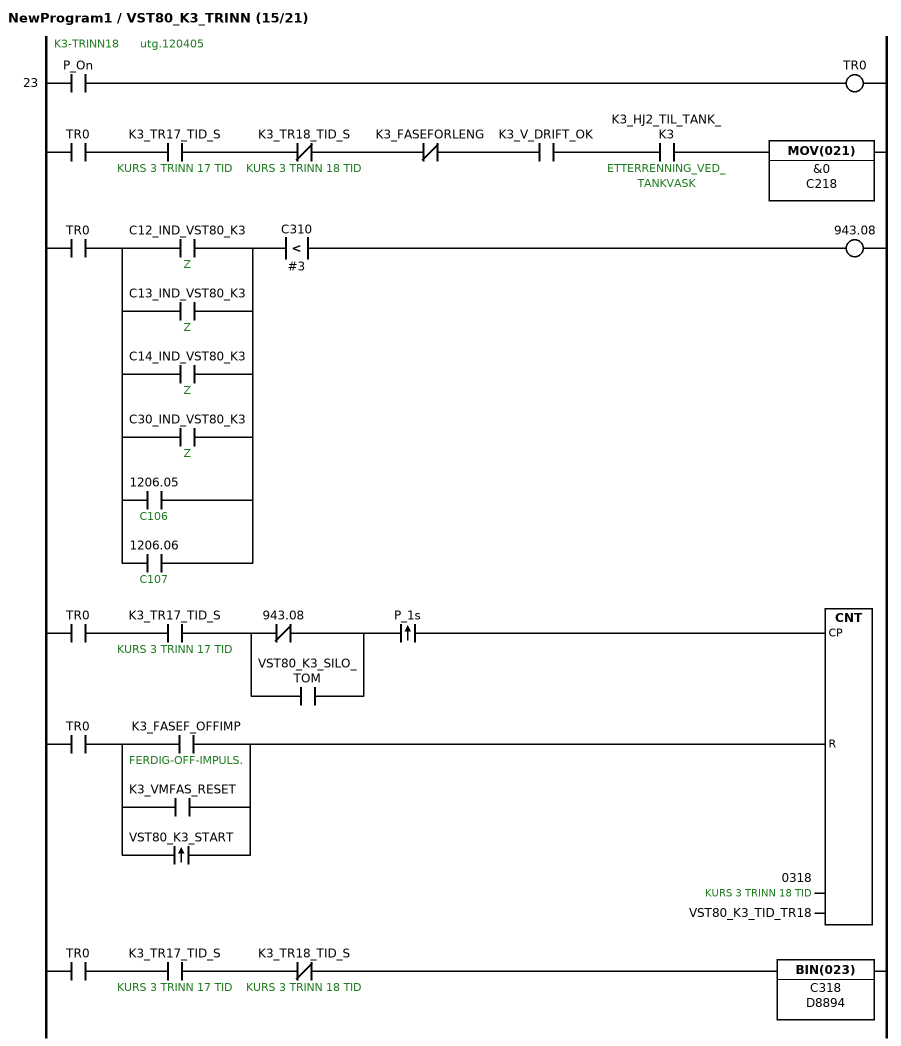
; [picture p336: NewProgram1 / VST80_K3_TRINN, rungs 23-23]
; rung 23: K3-TRINN18      utg.120405
LD P_On
OUT TR0
AND K3_TR17_TID_S  ; KURS 3 TRINN 17 TID
ANDNOT K3_TR18_TID_S  ; KURS 3 TRINN 18 TID
ANDNOT K3_FASEFORLENG
AND K3_V_DRIFT_OK
AND K3_HJ2_TIL_TANK_K3  ; ETTERRENNING_VED_TANKVASK
MOV(021) &0 C218
LD TR0
LD C12_IND_VST80_K3  ; Z
OR C13_IND_VST80_K3  ; Z
OR C14_IND_VST80_K3  ; Z
OR C30_IND_VST80_K3  ; Z
OR 1206.05  ; C106
OR 1206.06  ; C107
ANDLD
AND<(310) C310 #3
OUT 943.08
LD TR0
AND K3_TR17_TID_S  ; KURS 3 TRINN 17 TID
LDNOT 943.08
OR VST80_K3_SILO_TOM
ANDLD
@AND P_1s
LD TR0
LD K3_FASEF_OFFIMP  ; FERDIG-OFF-IMPULS.
OR K3_VMFAS_RESET
@OR VST80_K3_START
ANDLD
CNT 0318 VST80_K3_TID_TR18  ; KURS 3 TRINN 18 TID
LD TR0
AND K3_TR17_TID_S  ; KURS 3 TRINN 17 TID
ANDNOT K3_TR18_TID_S  ; KURS 3 TRINN 18 TID
BIN(023) C318 D8894

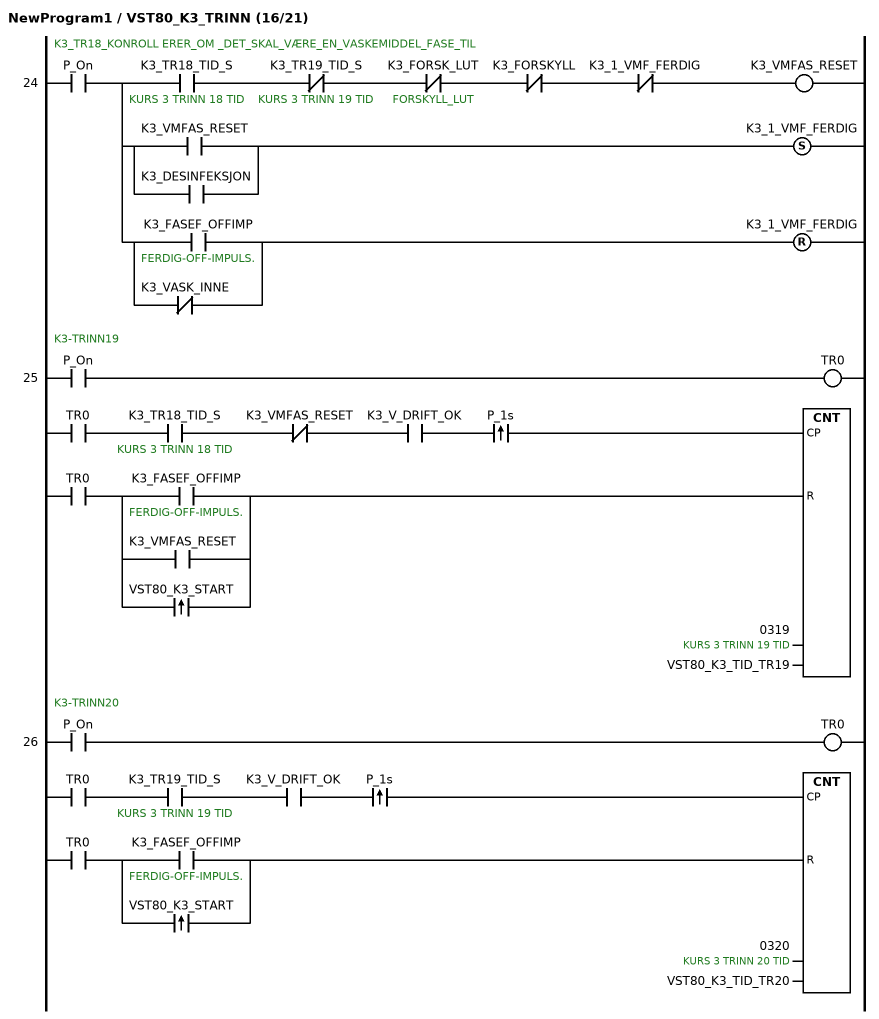
; rung 24: K3_TR18_KONROLL ERER_OM_DET_SKAL_VÆRE_EN_VASKEMIDDEL_FASE_TIL
LD P_On
OUT TR0
AND K3_TR18_TID_S  ; KURS 3 TRINN 18 TID
ANDNOT K3_TR19_TID_S  ; KURS 3 TRINN 19 TID
ANDNOT K3_FORSK_LUT  ; FORSKYLL_LUT
ANDNOT K3_FORSKYLL
ANDNOT K3_1_VMF_FERDIG
OUT K3_VMFAS_RESET
LD TR0
LD K3_VMFAS_RESET
OR K3_DESINFEKSJON
ANDLD
SET K3_1_VMF_FERDIG
LD TR0
LD K3_FASEF_OFFIMP  ; FERDIG-OFF-IMPULS.
ORNOT K3_VASK_INNE
ANDLD
RSET K3_1_VMF_FERDIG
; rung 25: K3-TRINN19
LD P_On
OUT TR0
AND K3_TR18_TID_S  ; KURS 3 TRINN 18 TID
ANDNOT K3_VMFAS_RESET
AND K3_V_DRIFT_OK
@AND P_1s
LD TR0
LD K3_FASEF_OFFIMP  ; FERDIG-OFF-IMPULS.
OR K3_VMFAS_RESET
@OR VST80_K3_START
ANDLD
CNT 0319 VST80_K3_TID_TR19  ; KURS 3 TRINN 19 TID
; rung 26: K3-TRINN20
LD P_On
OUT TR0
AND K3_TR19_TID_S  ; KURS 3 TRINN 19 TID
AND K3_V_DRIFT_OK
@AND P_1s
LD TR0
LD K3_FASEF_OFFIMP  ; FERDIG-OFF-IMPULS.
@OR VST80_K3_START
ANDLD
CNT 0320 VST80_K3_TID_TR20  ; KURS 3 TRINN 20 TID

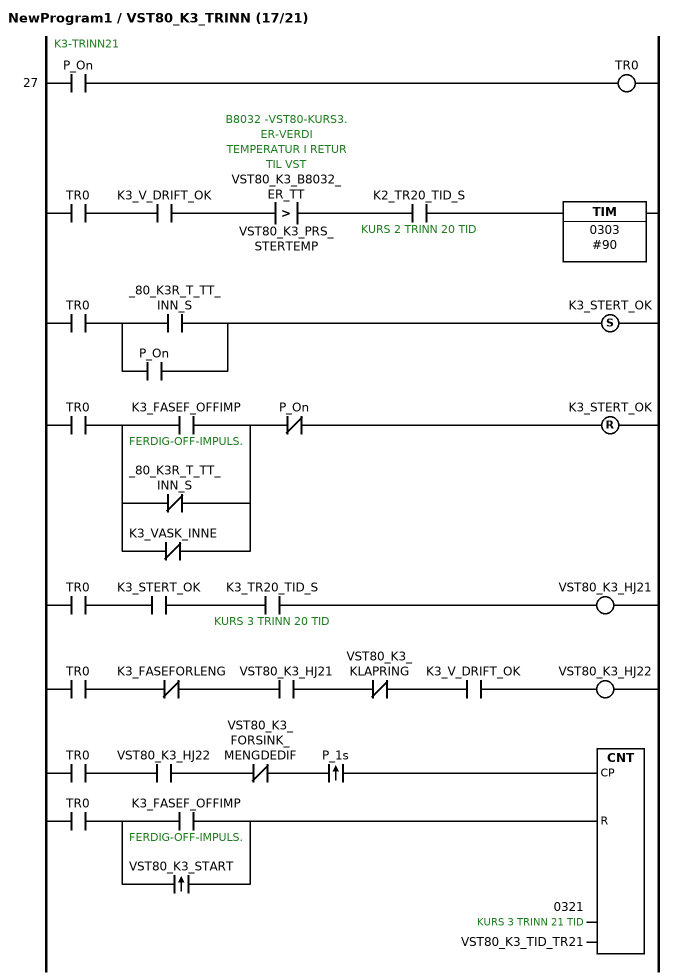
; rung 27: K3-TRINN21
LD P_On
OUT TR0
AND K3_V_DRIFT_OK
AND>(320) VST80_K3_B8032_ER_TT VST80_K3_PRS_STERTEMP  ; B8032 -VST80-KURS3. ER-VERDI TEMPERATUR I RETUR TIL VST
AND K2_TR20_TID_S  ; KURS 2 TRINN 20 TID
TIM 0303 #90
LD TR0
LD _80_K3R_T_TT_INN_S
OR P_On
ANDLD
SET K3_STERT_OK
LD TR0
LD K3_FASEF_OFFIMP  ; FERDIG-OFF-IMPULS.
ORNOT _80_K3R_T_TT_INN_S
ORNOT K3_VASK_INNE
ANDLD
ANDNOT P_On
RSET K3_STERT_OK
LD TR0
AND K3_STERT_OK
AND K3_TR20_TID_S  ; KURS 3 TRINN 20 TID
OUT VST80_K3_HJ21
LD TR0
ANDNOT K3_FASEFORLENG
AND VST80_K3_HJ21
ANDNOT VST80_K3_KLAPRING
AND K3_V_DRIFT_OK
OUT VST80_K3_HJ22
LD TR0
AND VST80_K3_HJ22
ANDNOT VST80_K3_FORSINK_MENGDEDIF
@AND P_1s
LD TR0
LD K3_FASEF_OFFIMP  ; FERDIG-OFF-IMPULS.
@OR VST80_K3_START
ANDLD
CNT 0321 VST80_K3_TID_TR21  ; KURS 3 TRINN 21 TID

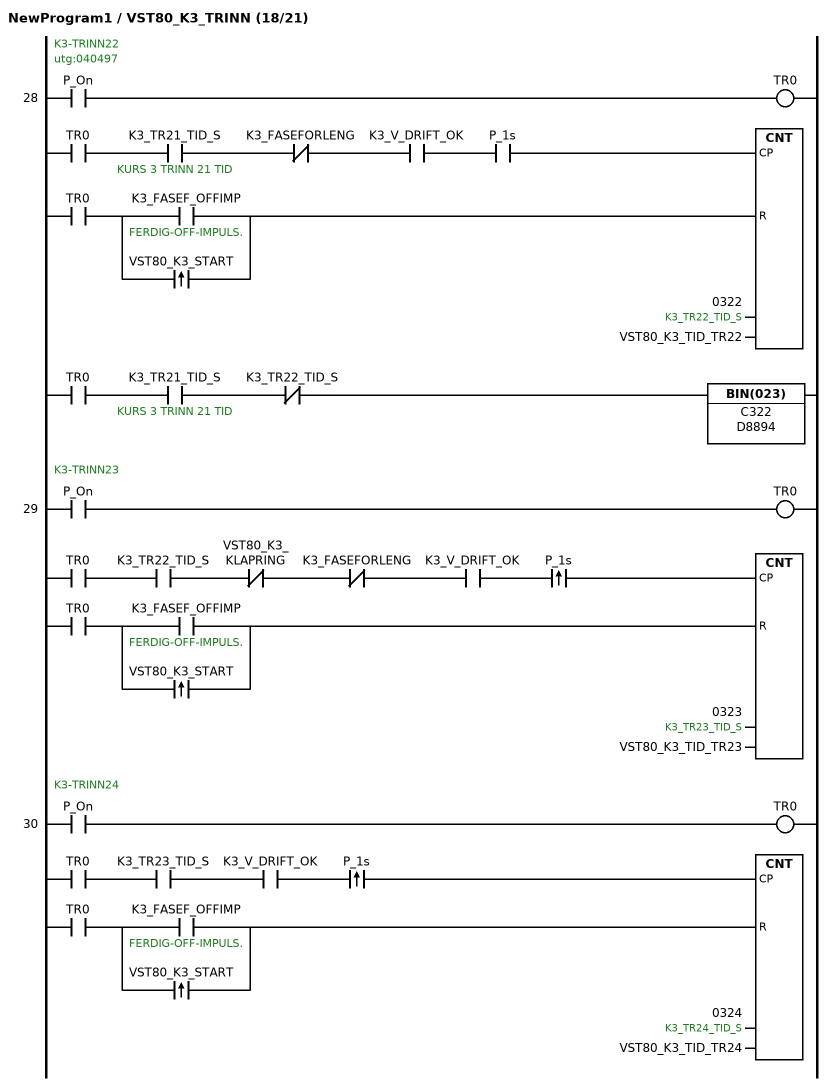
; rung 28: K3-TRINN22 / utg:040497
LD P_On
OUT TR0
AND K3_TR21_TID_S  ; KURS 3 TRINN 21 TID
ANDNOT K3_FASEFORLENG
AND K3_V_DRIFT_OK
AND P_1s
LD TR0
LD K3_FASEF_OFFIMP  ; FERDIG-OFF-IMPULS.
@OR VST80_K3_START
ANDLD
CNT 0322 VST80_K3_TID_TR22  ; K3_TR22_TID_S
LD TR0
AND K3_TR21_TID_S  ; KURS 3 TRINN 21 TID
ANDNOT K3_TR22_TID_S
BIN(023) C322 D8894
; rung 29: K3-TRINN23
LD P_On
OUT TR0
AND K3_TR22_TID_S
ANDNOT VST80_K3_KLAPRING
ANDNOT K3_FASEFORLENG
AND K3_V_DRIFT_OK
@AND P_1s
LD TR0
LD K3_FASEF_OFFIMP  ; FERDIG-OFF-IMPULS.
@OR VST80_K3_START
ANDLD
CNT 0323 VST80_K3_TID_TR23  ; K3_TR23_TID_S
; rung 30: K3-TRINN24
LD P_On
OUT TR0
AND K3_TR23_TID_S
AND K3_V_DRIFT_OK
@AND P_1s
LD TR0
LD K3_FASEF_OFFIMP  ; FERDIG-OFF-IMPULS.
@OR VST80_K3_START
ANDLD
CNT 0324 VST80_K3_TID_TR24  ; K3_TR24_TID_S

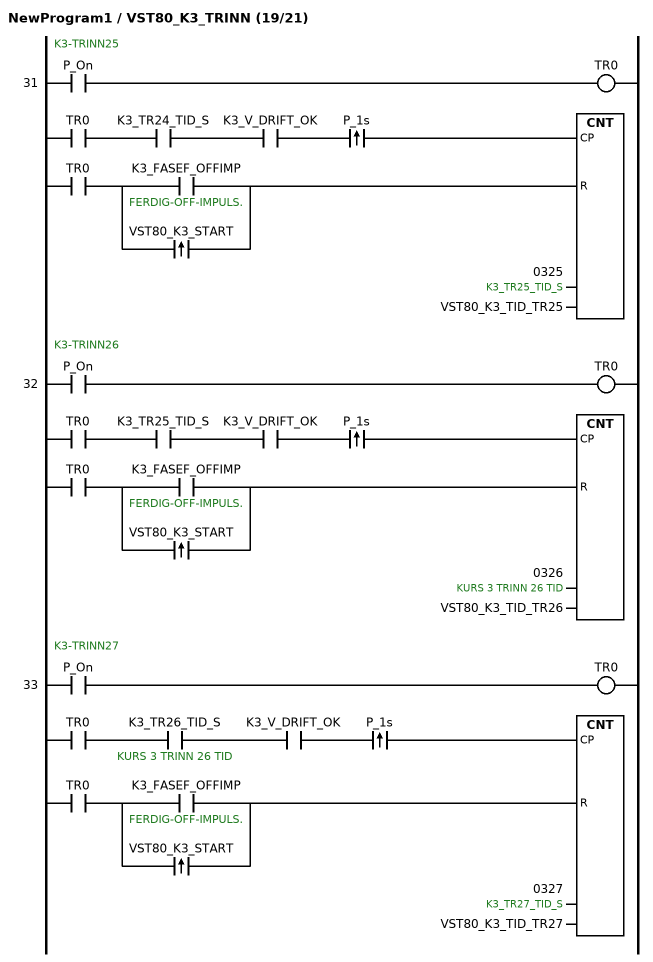
; rung 31: K3-TRINN25
LD P_On
OUT TR0
AND K3_TR24_TID_S
AND K3_V_DRIFT_OK
@AND P_1s
LD TR0
LD K3_FASEF_OFFIMP  ; FERDIG-OFF-IMPULS.
@OR VST80_K3_START
ANDLD
CNT 0325 VST80_K3_TID_TR25  ; K3_TR25_TID_S
; rung 32: K3-TRINN26
LD P_On
OUT TR0
AND K3_TR25_TID_S
AND K3_V_DRIFT_OK
@AND P_1s
LD TR0
LD K3_FASEF_OFFIMP  ; FERDIG-OFF-IMPULS.
@OR VST80_K3_START
ANDLD
CNT 0326 VST80_K3_TID_TR26  ; KURS 3 TRINN 26 TID
; rung 33: K3-TRINN27
LD P_On
OUT TR0
AND K3_TR26_TID_S  ; KURS 3 TRINN 26 TID
AND K3_V_DRIFT_OK
@AND P_1s
LD TR0
LD K3_FASEF_OFFIMP  ; FERDIG-OFF-IMPULS.
@OR VST80_K3_START
ANDLD
CNT 0327 VST80_K3_TID_TR27  ; K3_TR27_TID_S

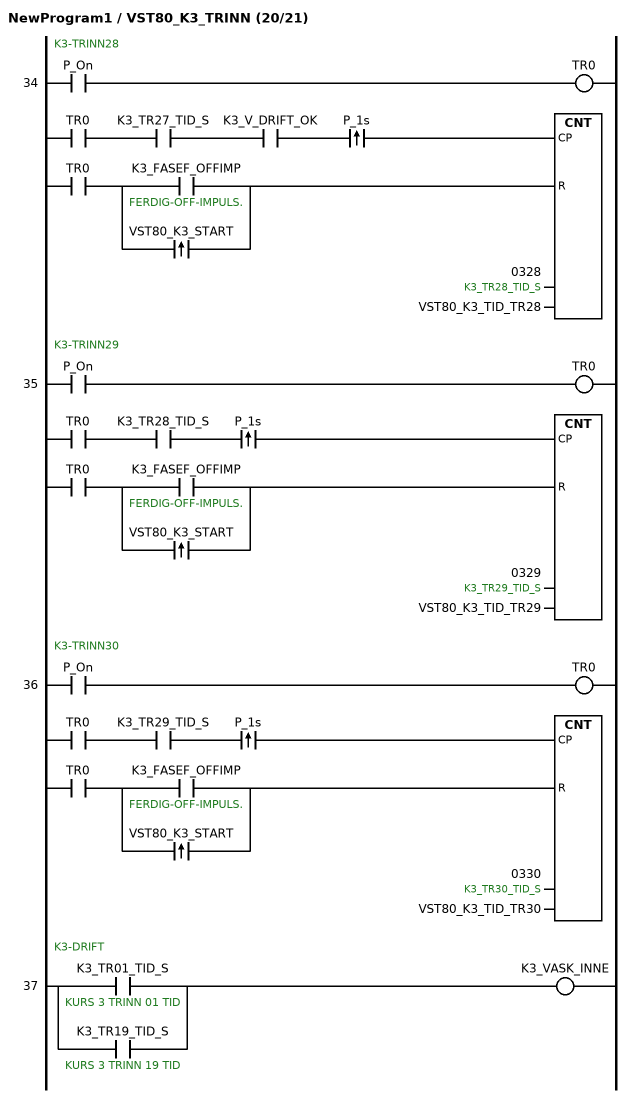
; rung 34: K3-TRINN28
LD P_On
OUT TR0
AND K3_TR27_TID_S
AND K3_V_DRIFT_OK
@AND P_1s
LD TR0
LD K3_FASEF_OFFIMP  ; FERDIG-OFF-IMPULS.
@OR VST80_K3_START
ANDLD
CNT 0328 VST80_K3_TID_TR28  ; K3_TR28_TID_S
; rung 35: K3-TRINN29
LD P_On
OUT TR0
AND K3_TR28_TID_S
@AND P_1s
LD TR0
LD K3_FASEF_OFFIMP  ; FERDIG-OFF-IMPULS.
@OR VST80_K3_START
ANDLD
CNT 0329 VST80_K3_TID_TR29  ; K3_TR29_TID_S
; rung 36: K3-TRINN30
LD P_On
OUT TR0
AND K3_TR29_TID_S
@AND P_1s
LD TR0
LD K3_FASEF_OFFIMP  ; FERDIG-OFF-IMPULS.
@OR VST80_K3_START
ANDLD
CNT 0330 VST80_K3_TID_TR30  ; K3_TR30_TID_S
; rung 37: K3-DRIFT
LD K3_TR01_TID_S  ; KURS 3 TRINN 01 TID
OR K3_TR19_TID_S  ; KURS 3 TRINN 19 TID
OUT K3_VASK_INNE

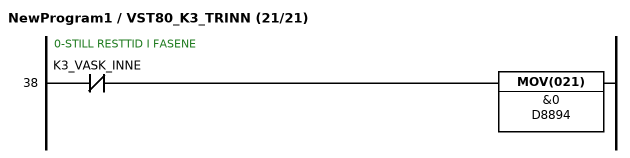
; rung 38: 0-STILL RESTTID I FASENE
LDNOT K3_VASK_INNE
MOV(021) &0 D8894

### Section VST80_K3_ANALOGSIGN_INN

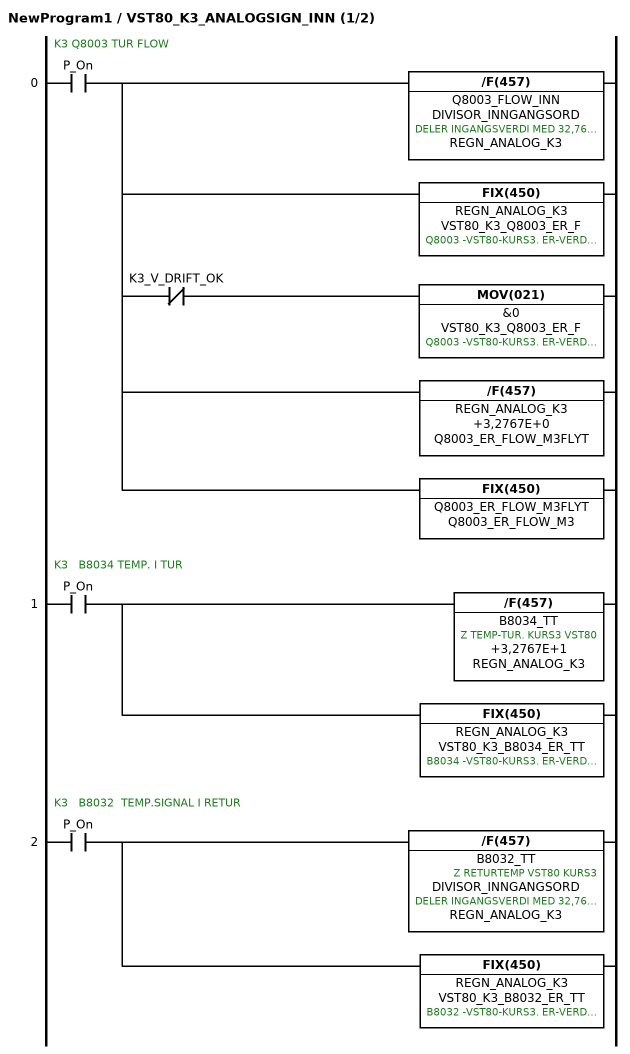
; rung 0: K3 Q8003 TUR FLOW
LD P_On
OUT TR0
/F(457) Q8003_FLOW_INN DIVISOR_INNGANGSORD REGN_ANALOG_K3  ; DELER INGANGSVERDI MED 32,760 FOR OMREGNING TIL 0-1000
FIX(450) REGN_ANALOG_K3 VST80_K3_Q8003_ER_F  ; Q8003 -VST80-KURS3. ER-VERDI FLOW I TUR
ANDNOT K3_V_DRIFT_OK
MOV(021) &0 VST80_K3_Q8003_ER_F  ; Q8003 -VST80-KURS3. ER-VERDI FLOW I TUR
LD TR0
/F(457) REGN_ANALOG_K3 +3,2767E+0 Q8003_ER_FLOW_M3FLYT
FIX(450) Q8003_ER_FLOW_M3FLYT Q8003_ER_FLOW_M3
; rung 1: K3   B8034 TEMP. I TUR
LD P_On
/F(457) B8034_TT +3,2767E+1 REGN_ANALOG_K3  ; Z TEMP-TUR. KURS3 VST80
FIX(450) REGN_ANALOG_K3 VST80_K3_B8034_ER_TT  ; B8034 -VST80-KURS3. ER-VERDI TEMPERATUR I TUR TIL VST
; rung 2: K3   B8032  TEMP.SIGNAL I RETUR
LD P_On
/F(457) B8032_TT DIVISOR_INNGANGSORD REGN_ANALOG_K3  ; Z RETURTEMP VST80 KURS3, DELER INGANGSVERDI MED 32,760 FOR OMREGNING TIL 0-1000
FIX(450) REGN_ANALOG_K3 VST80_K3_B8032_ER_TT  ; B8032 -VST80-KURS3. ER-VERDI TEMPERATUR I RETUR TIL VST

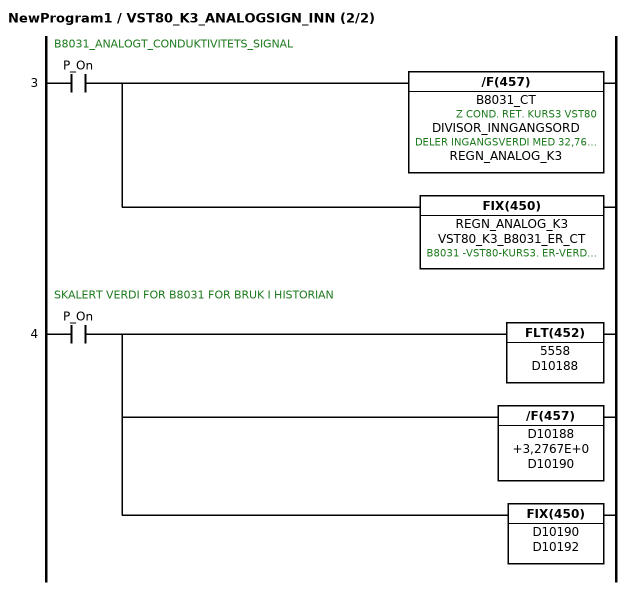
; rung 3: B8031_ANALOGT_CONDUKTIVITETS_SIGNAL
LD P_On
/F(457) B8031_CT DIVISOR_INNGANGSORD REGN_ANALOG_K3  ; Z COND. RET. KURS3 VST80, DELER INGANGSVERDI MED 32,760 FOR OMREGNING TIL 0-1000
FIX(450) REGN_ANALOG_K3 VST80_K3_B8031_ER_CT  ; B8031 -VST80-KURS3. ER-VERDI KONDUKTIVITET I RETUR TIL VST
; rung 4: SKALERT VERDI FOR B8031 FOR BRUK I HISTORIAN
LD P_On
FLT(452) 5558 D10188
/F(457) D10188 +3,2767E+0 D10190
FIX(450) D10190 D10192

### Section VST_80_K3_TYPE_VASK
; KOMMANDOGIVNING FOR VALG AV TYPE VASK. / 2: DESINFEKSJON / 3: FORSKYLL

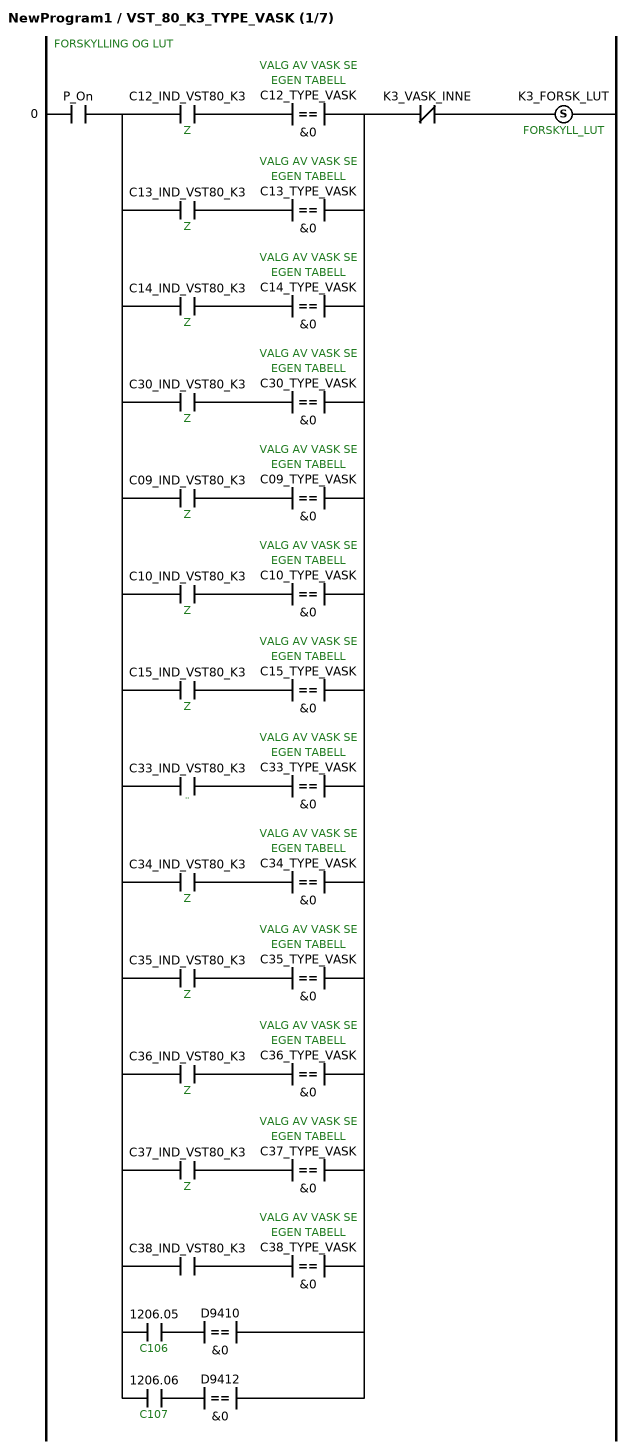
; rung 0: FORSKYLLING OG LUT
LD P_On
LD C12_IND_VST80_K3  ; Z
AND=(300) C12_TYPE_VASK &0  ; VALG AV VASK SE EGEN TABELL
LD C13_IND_VST80_K3  ; Z
AND=(300) C13_TYPE_VASK &0  ; VALG AV VASK SE EGEN TABELL
ORLD
LD C14_IND_VST80_K3  ; Z
AND=(300) C14_TYPE_VASK &0  ; VALG AV VASK SE EGEN TABELL
ORLD
LD C30_IND_VST80_K3  ; Z
AND=(300) C30_TYPE_VASK &0  ; VALG AV VASK SE EGEN TABELL
ORLD
LD C09_IND_VST80_K3  ; Z
AND=(300) C09_TYPE_VASK &0  ; VALG AV VASK SE EGEN TABELL
ORLD
LD C10_IND_VST80_K3  ; Z
AND=(300) C10_TYPE_VASK &0  ; VALG AV VASK SE EGEN TABELL
ORLD
LD C15_IND_VST80_K3  ; Z
AND=(300) C15_TYPE_VASK &0  ; VALG AV VASK SE EGEN TABELL
ORLD
LD C33_IND_VST80_K3  ; ¨
AND=(300) C33_TYPE_VASK &0  ; VALG AV VASK SE EGEN TABELL
ORLD
LD C34_IND_VST80_K3  ; Z
AND=(300) C34_TYPE_VASK &0  ; VALG AV VASK SE EGEN TABELL
ORLD
LD C35_IND_VST80_K3  ; Z
AND=(300) C35_TYPE_VASK &0  ; VALG AV VASK SE EGEN TABELL
ORLD
LD C36_IND_VST80_K3  ; Z
AND=(300) C36_TYPE_VASK &0  ; VALG AV VASK SE EGEN TABELL
ORLD
LD C37_IND_VST80_K3  ; Z
AND=(300) C37_TYPE_VASK &0  ; VALG AV VASK SE EGEN TABELL
ORLD
LD C38_IND_VST80_K3
AND=(300) C38_TYPE_VASK &0  ; VALG AV VASK SE EGEN TABELL
ORLD
LD 1206.05  ; C106
AND=(300) D9410 &0
ORLD
LD 1206.06  ; C107
AND=(300) D9412 &0
ORLD
ANDLD
ANDNOT K3_VASK_INNE
SET K3_FORSK_LUT  ; FORSKYLL_LUT

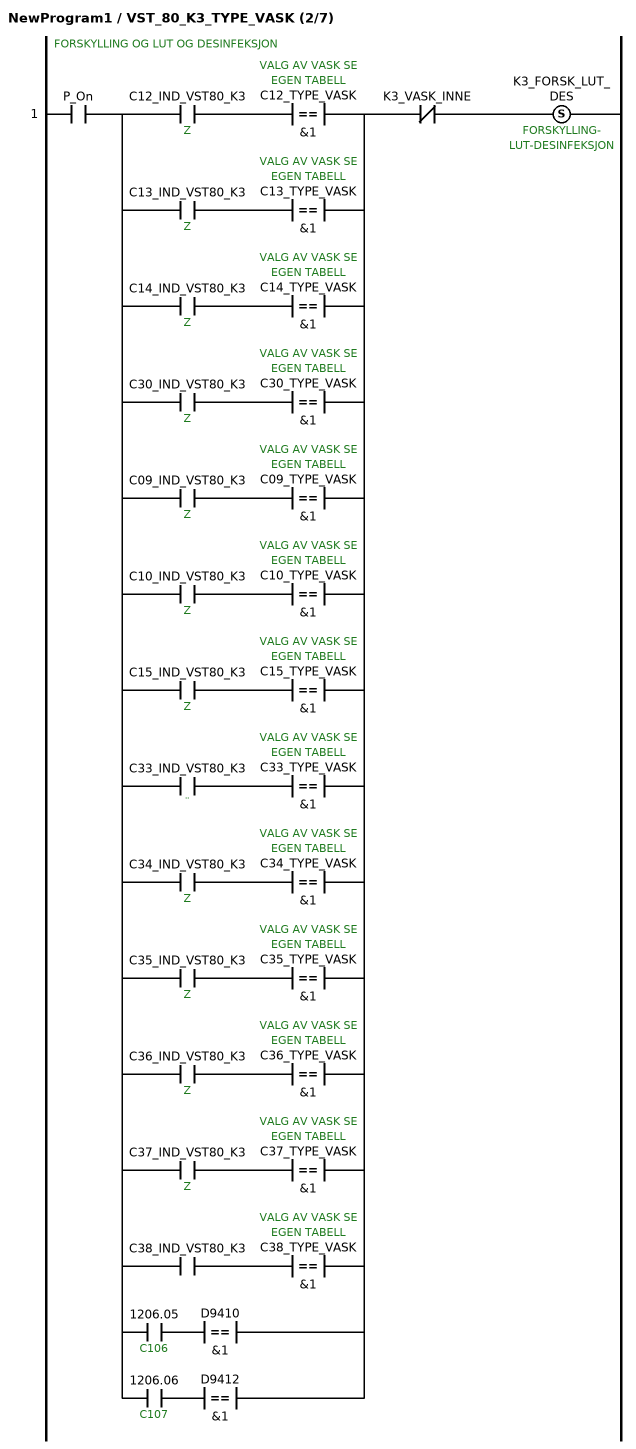
; rung 1: FORSKYLLING OG LUT OG DESINFEKSJON
LD P_On
LD C12_IND_VST80_K3  ; Z
AND=(300) C12_TYPE_VASK &1  ; VALG AV VASK SE EGEN TABELL
LD C13_IND_VST80_K3  ; Z
AND=(300) C13_TYPE_VASK &1  ; VALG AV VASK SE EGEN TABELL
ORLD
LD C14_IND_VST80_K3  ; Z
AND=(300) C14_TYPE_VASK &1  ; VALG AV VASK SE EGEN TABELL
ORLD
LD C30_IND_VST80_K3  ; Z
AND=(300) C30_TYPE_VASK &1  ; VALG AV VASK SE EGEN TABELL
ORLD
LD C09_IND_VST80_K3  ; Z
AND=(300) C09_TYPE_VASK &1  ; VALG AV VASK SE EGEN TABELL
ORLD
LD C10_IND_VST80_K3  ; Z
AND=(300) C10_TYPE_VASK &1  ; VALG AV VASK SE EGEN TABELL
ORLD
LD C15_IND_VST80_K3  ; Z
AND=(300) C15_TYPE_VASK &1  ; VALG AV VASK SE EGEN TABELL
ORLD
LD C33_IND_VST80_K3  ; ¨
AND=(300) C33_TYPE_VASK &1  ; VALG AV VASK SE EGEN TABELL
ORLD
LD C34_IND_VST80_K3  ; Z
AND=(300) C34_TYPE_VASK &1  ; VALG AV VASK SE EGEN TABELL
ORLD
LD C35_IND_VST80_K3  ; Z
AND=(300) C35_TYPE_VASK &1  ; VALG AV VASK SE EGEN TABELL
ORLD
LD C36_IND_VST80_K3  ; Z
AND=(300) C36_TYPE_VASK &1  ; VALG AV VASK SE EGEN TABELL
ORLD
LD C37_IND_VST80_K3  ; Z
AND=(300) C37_TYPE_VASK &1  ; VALG AV VASK SE EGEN TABELL
ORLD
LD C38_IND_VST80_K3
AND=(300) C38_TYPE_VASK &1  ; VALG AV VASK SE EGEN TABELL
ORLD
LD 1206.05  ; C106
AND=(300) D9410 &1
ORLD
LD 1206.06  ; C107
AND=(300) D9412 &1
ORLD
ANDLD
ANDNOT K3_VASK_INNE
SET K3_FORSK_LUT_DES  ; FORSKYLLING- LUT-DESINFEKSJON

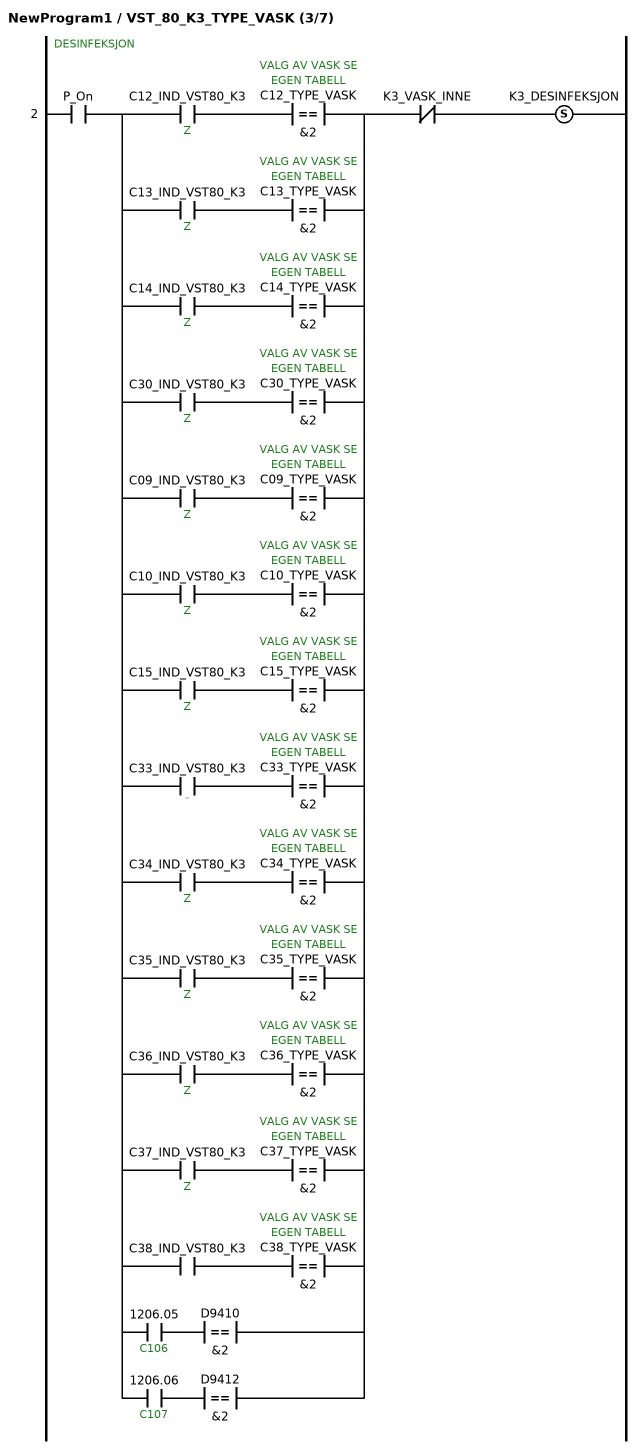
; rung 2: DESINFEKSJON
LD P_On
LD C12_IND_VST80_K3  ; Z
AND=(300) C12_TYPE_VASK &2  ; VALG AV VASK SE EGEN TABELL
LD C13_IND_VST80_K3  ; Z
AND=(300) C13_TYPE_VASK &2  ; VALG AV VASK SE EGEN TABELL
ORLD
LD C14_IND_VST80_K3  ; Z
AND=(300) C14_TYPE_VASK &2  ; VALG AV VASK SE EGEN TABELL
ORLD
LD C30_IND_VST80_K3  ; Z
AND=(300) C30_TYPE_VASK &2  ; VALG AV VASK SE EGEN TABELL
ORLD
LD C09_IND_VST80_K3  ; Z
AND=(300) C09_TYPE_VASK &2  ; VALG AV VASK SE EGEN TABELL
ORLD
LD C10_IND_VST80_K3  ; Z
AND=(300) C10_TYPE_VASK &2  ; VALG AV VASK SE EGEN TABELL
ORLD
LD C15_IND_VST80_K3  ; Z
AND=(300) C15_TYPE_VASK &2  ; VALG AV VASK SE EGEN TABELL
ORLD
LD C33_IND_VST80_K3  ; ¨
AND=(300) C33_TYPE_VASK &2  ; VALG AV VASK SE EGEN TABELL
ORLD
LD C34_IND_VST80_K3  ; Z
AND=(300) C34_TYPE_VASK &2  ; VALG AV VASK SE EGEN TABELL
ORLD
LD C35_IND_VST80_K3  ; Z
AND=(300) C35_TYPE_VASK &2  ; VALG AV VASK SE EGEN TABELL
ORLD
LD C36_IND_VST80_K3  ; Z
AND=(300) C36_TYPE_VASK &2  ; VALG AV VASK SE EGEN TABELL
ORLD
LD C37_IND_VST80_K3  ; Z
AND=(300) C37_TYPE_VASK &2  ; VALG AV VASK SE EGEN TABELL
ORLD
LD C38_IND_VST80_K3
AND=(300) C38_TYPE_VASK &2  ; VALG AV VASK SE EGEN TABELL
ORLD
LD 1206.05  ; C106
AND=(300) D9410 &2
ORLD
LD 1206.06  ; C107
AND=(300) D9412 &2
ORLD
ANDLD
ANDNOT K3_VASK_INNE
SET K3_DESINFEKSJON

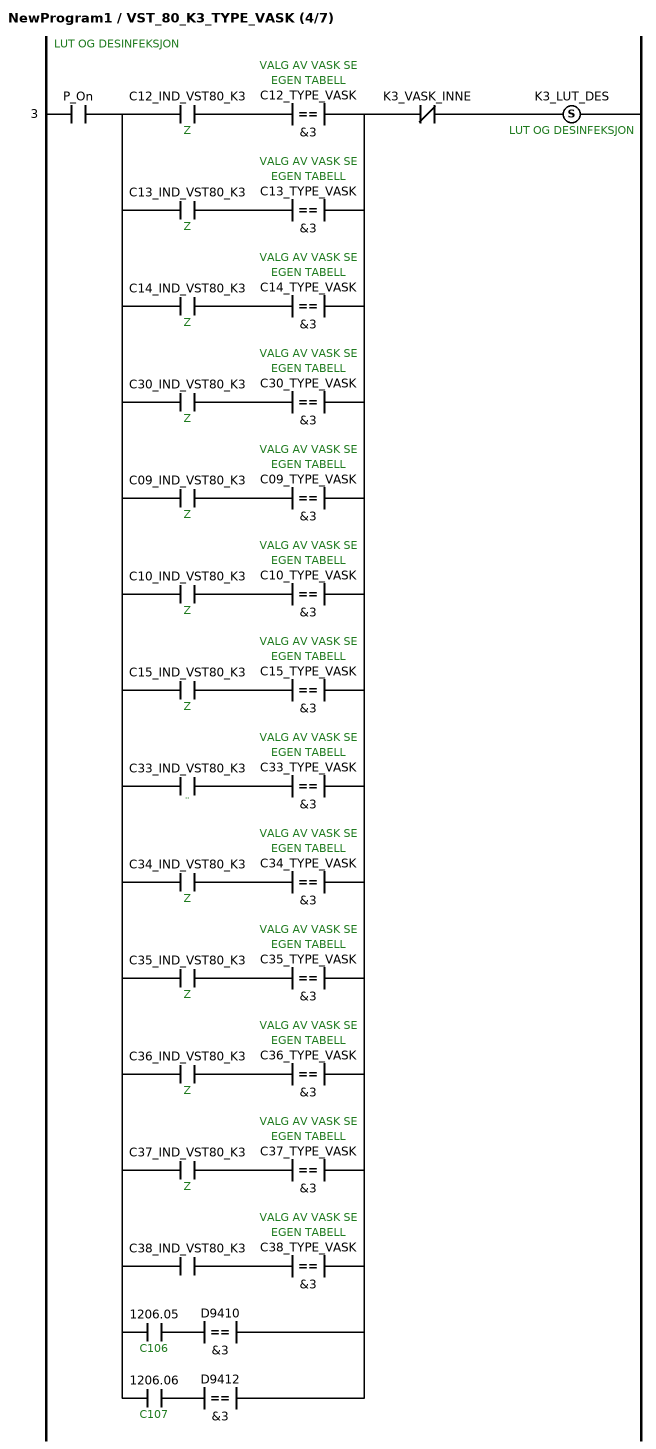
; rung 3: LUT OG DESINFEKSJON
LD P_On
LD C12_IND_VST80_K3  ; Z
AND=(300) C12_TYPE_VASK &3  ; VALG AV VASK SE EGEN TABELL
LD C13_IND_VST80_K3  ; Z
AND=(300) C13_TYPE_VASK &3  ; VALG AV VASK SE EGEN TABELL
ORLD
LD C14_IND_VST80_K3  ; Z
AND=(300) C14_TYPE_VASK &3  ; VALG AV VASK SE EGEN TABELL
ORLD
LD C30_IND_VST80_K3  ; Z
AND=(300) C30_TYPE_VASK &3  ; VALG AV VASK SE EGEN TABELL
ORLD
LD C09_IND_VST80_K3  ; Z
AND=(300) C09_TYPE_VASK &3  ; VALG AV VASK SE EGEN TABELL
ORLD
LD C10_IND_VST80_K3  ; Z
AND=(300) C10_TYPE_VASK &3  ; VALG AV VASK SE EGEN TABELL
ORLD
LD C15_IND_VST80_K3  ; Z
AND=(300) C15_TYPE_VASK &3  ; VALG AV VASK SE EGEN TABELL
ORLD
LD C33_IND_VST80_K3  ; ¨
AND=(300) C33_TYPE_VASK &3  ; VALG AV VASK SE EGEN TABELL
ORLD
LD C34_IND_VST80_K3  ; Z
AND=(300) C34_TYPE_VASK &3  ; VALG AV VASK SE EGEN TABELL
ORLD
LD C35_IND_VST80_K3  ; Z
AND=(300) C35_TYPE_VASK &3  ; VALG AV VASK SE EGEN TABELL
ORLD
LD C36_IND_VST80_K3  ; Z
AND=(300) C36_TYPE_VASK &3  ; VALG AV VASK SE EGEN TABELL
ORLD
LD C37_IND_VST80_K3  ; Z
AND=(300) C37_TYPE_VASK &3  ; VALG AV VASK SE EGEN TABELL
ORLD
LD C38_IND_VST80_K3
AND=(300) C38_TYPE_VASK &3  ; VALG AV VASK SE EGEN TABELL
ORLD
LD 1206.05  ; C106
AND=(300) D9410 &3
ORLD
LD 1206.06  ; C107
AND=(300) D9412 &3
ORLD
ANDLD
ANDNOT K3_VASK_INNE
SET K3_LUT_DES  ; LUT OG DESINFEKSJON

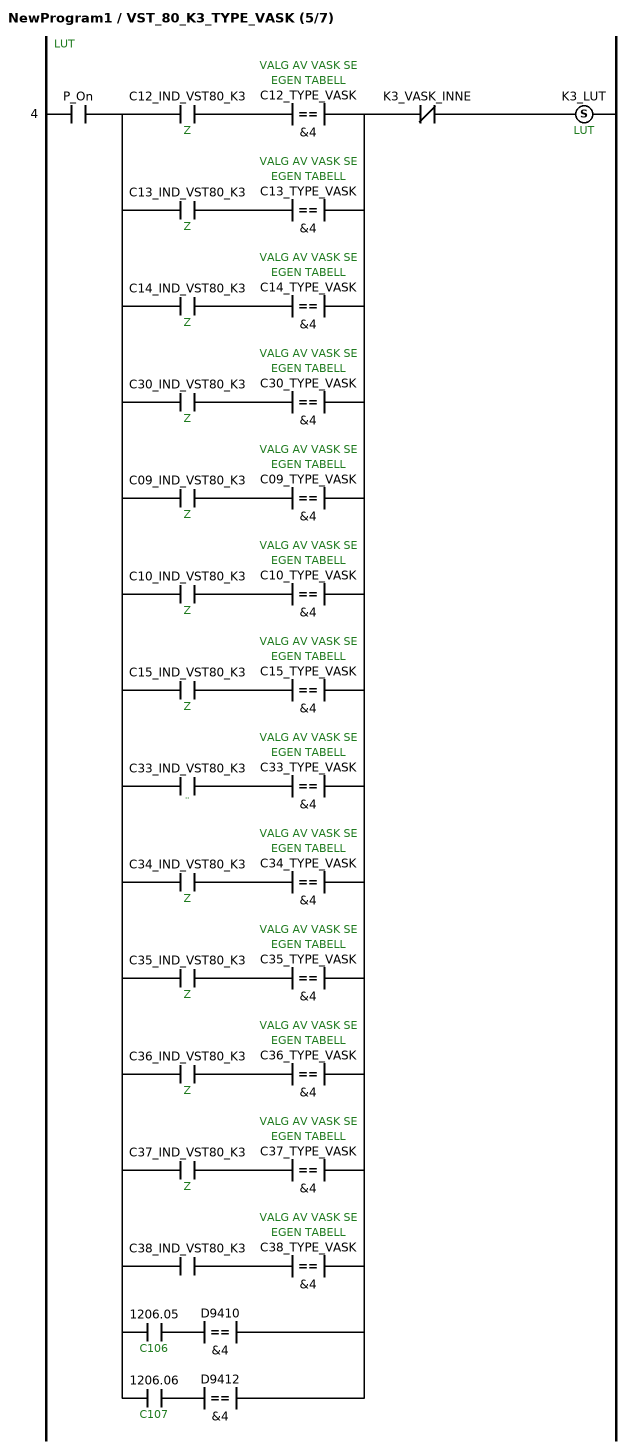
; rung 4: LUT
LD P_On
LD C12_IND_VST80_K3  ; Z
AND=(300) C12_TYPE_VASK &4  ; VALG AV VASK SE EGEN TABELL
LD C13_IND_VST80_K3  ; Z
AND=(300) C13_TYPE_VASK &4  ; VALG AV VASK SE EGEN TABELL
ORLD
LD C14_IND_VST80_K3  ; Z
AND=(300) C14_TYPE_VASK &4  ; VALG AV VASK SE EGEN TABELL
ORLD
LD C30_IND_VST80_K3  ; Z
AND=(300) C30_TYPE_VASK &4  ; VALG AV VASK SE EGEN TABELL
ORLD
LD C09_IND_VST80_K3  ; Z
AND=(300) C09_TYPE_VASK &4  ; VALG AV VASK SE EGEN TABELL
ORLD
LD C10_IND_VST80_K3  ; Z
AND=(300) C10_TYPE_VASK &4  ; VALG AV VASK SE EGEN TABELL
ORLD
LD C15_IND_VST80_K3  ; Z
AND=(300) C15_TYPE_VASK &4  ; VALG AV VASK SE EGEN TABELL
ORLD
LD C33_IND_VST80_K3  ; ¨
AND=(300) C33_TYPE_VASK &4  ; VALG AV VASK SE EGEN TABELL
ORLD
LD C34_IND_VST80_K3  ; Z
AND=(300) C34_TYPE_VASK &4  ; VALG AV VASK SE EGEN TABELL
ORLD
LD C35_IND_VST80_K3  ; Z
AND=(300) C35_TYPE_VASK &4  ; VALG AV VASK SE EGEN TABELL
ORLD
LD C36_IND_VST80_K3  ; Z
AND=(300) C36_TYPE_VASK &4  ; VALG AV VASK SE EGEN TABELL
ORLD
LD C37_IND_VST80_K3  ; Z
AND=(300) C37_TYPE_VASK &4  ; VALG AV VASK SE EGEN TABELL
ORLD
LD C38_IND_VST80_K3
AND=(300) C38_TYPE_VASK &4  ; VALG AV VASK SE EGEN TABELL
ORLD
LD 1206.05  ; C106
AND=(300) D9410 &4
ORLD
LD 1206.06  ; C107
AND=(300) D9412 &4
ORLD
ANDLD
ANDNOT K3_VASK_INNE
SET K3_LUT  ; LUT

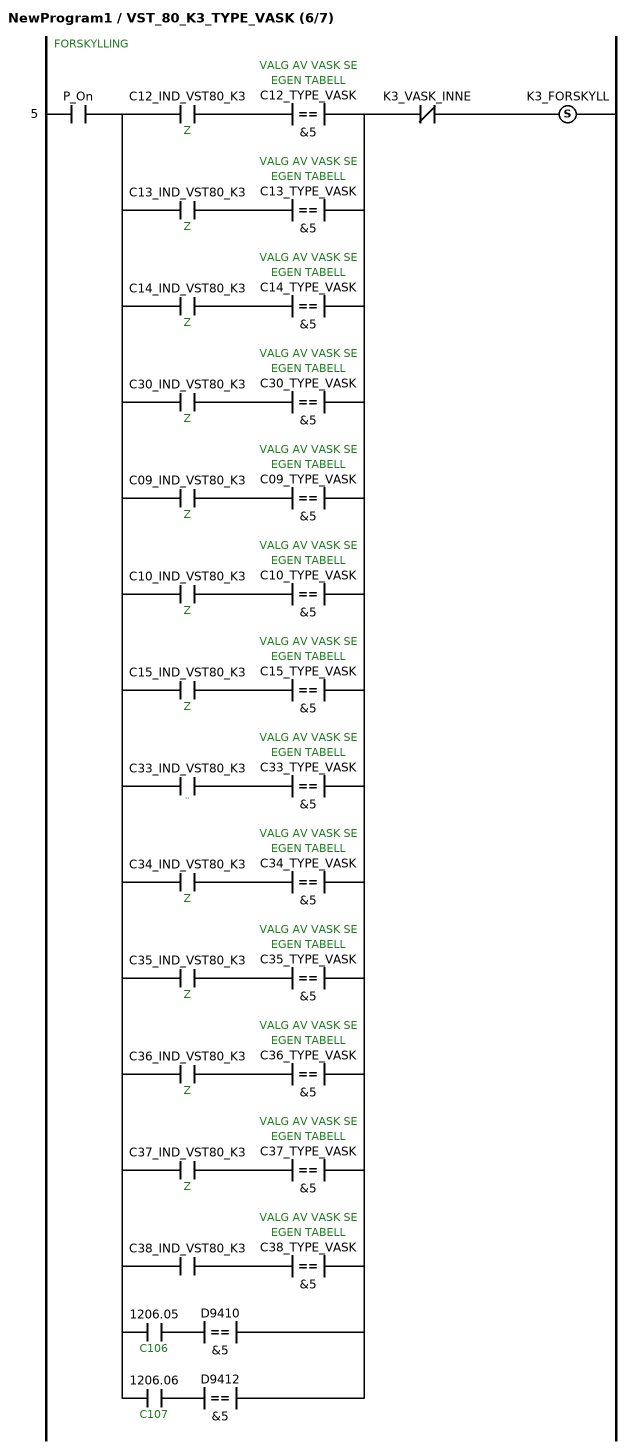
; rung 5: FORSKYLLING
LD P_On
LD C12_IND_VST80_K3  ; Z
AND=(300) C12_TYPE_VASK &5  ; VALG AV VASK SE EGEN TABELL
LD C13_IND_VST80_K3  ; Z
AND=(300) C13_TYPE_VASK &5  ; VALG AV VASK SE EGEN TABELL
ORLD
LD C14_IND_VST80_K3  ; Z
AND=(300) C14_TYPE_VASK &5  ; VALG AV VASK SE EGEN TABELL
ORLD
LD C30_IND_VST80_K3  ; Z
AND=(300) C30_TYPE_VASK &5  ; VALG AV VASK SE EGEN TABELL
ORLD
LD C09_IND_VST80_K3  ; Z
AND=(300) C09_TYPE_VASK &5  ; VALG AV VASK SE EGEN TABELL
ORLD
LD C10_IND_VST80_K3  ; Z
AND=(300) C10_TYPE_VASK &5  ; VALG AV VASK SE EGEN TABELL
ORLD
LD C15_IND_VST80_K3  ; Z
AND=(300) C15_TYPE_VASK &5  ; VALG AV VASK SE EGEN TABELL
ORLD
LD C33_IND_VST80_K3  ; ¨
AND=(300) C33_TYPE_VASK &5  ; VALG AV VASK SE EGEN TABELL
ORLD
LD C34_IND_VST80_K3  ; Z
AND=(300) C34_TYPE_VASK &5  ; VALG AV VASK SE EGEN TABELL
ORLD
LD C35_IND_VST80_K3  ; Z
AND=(300) C35_TYPE_VASK &5  ; VALG AV VASK SE EGEN TABELL
ORLD
LD C36_IND_VST80_K3  ; Z
AND=(300) C36_TYPE_VASK &5  ; VALG AV VASK SE EGEN TABELL
ORLD
LD C37_IND_VST80_K3  ; Z
AND=(300) C37_TYPE_VASK &5  ; VALG AV VASK SE EGEN TABELL
ORLD
LD C38_IND_VST80_K3
AND=(300) C38_TYPE_VASK &5  ; VALG AV VASK SE EGEN TABELL
ORLD
LD 1206.05  ; C106
AND=(300) D9410 &5
ORLD
LD 1206.06  ; C107
AND=(300) D9412 &5
ORLD
ANDLD
ANDNOT K3_VASK_INNE
SET K3_FORSKYLL

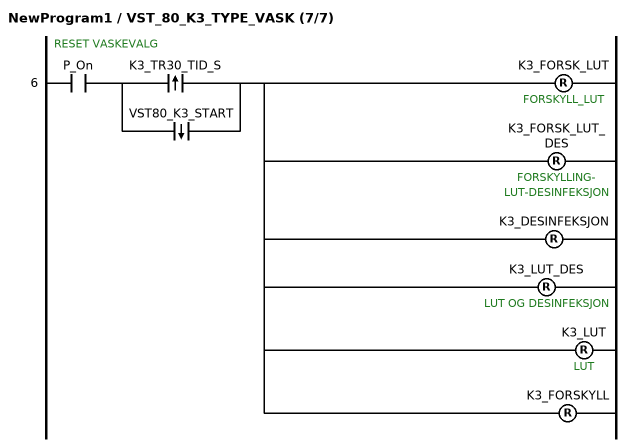
; rung 6: RESET VASKEVALG
LD P_On
@LD K3_TR30_TID_S
%OR VST80_K3_START
ANDLD
RSET K3_FORSK_LUT  ; FORSKYLL_LUT
RSET K3_FORSK_LUT_DES  ; FORSKYLLING- LUT-DESINFEKSJON
RSET K3_DESINFEKSJON
RSET K3_LUT_DES  ; LUT OG DESINFEKSJON
RSET K3_LUT  ; LUT
RSET K3_FORSKYLL

### Section VST80_K3_DR_STATUS

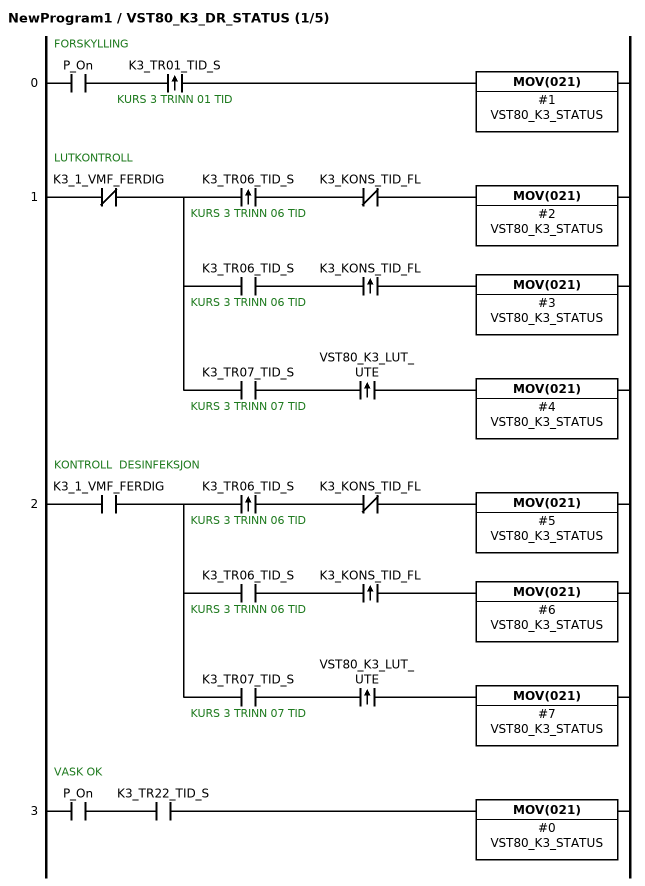
; rung 0: FORSKYLLING
LD P_On
@AND K3_TR01_TID_S  ; KURS 3 TRINN 01 TID
MOV(021) #1 VST80_K3_STATUS
; rung 1: LUTKONTROLL
LDNOT K3_1_VMF_FERDIG
OUT TR0
@AND K3_TR06_TID_S  ; KURS 3 TRINN 06 TID
ANDNOT K3_KONS_TID_FL
MOV(021) #2 VST80_K3_STATUS
LD TR0
AND K3_TR06_TID_S  ; KURS 3 TRINN 06 TID
@AND K3_KONS_TID_FL
MOV(021) #3 VST80_K3_STATUS
LD TR0
AND K3_TR07_TID_S  ; KURS 3 TRINN 07 TID
@AND VST80_K3_LUT_UTE
MOV(021) #4 VST80_K3_STATUS
; rung 2: KONTROLL  DESINFEKSJON
LD K3_1_VMF_FERDIG
OUT TR0
@AND K3_TR06_TID_S  ; KURS 3 TRINN 06 TID
ANDNOT K3_KONS_TID_FL
MOV(021) #5 VST80_K3_STATUS
LD TR0
AND K3_TR06_TID_S  ; KURS 3 TRINN 06 TID
@AND K3_KONS_TID_FL
MOV(021) #6 VST80_K3_STATUS
LD TR0
AND K3_TR07_TID_S  ; KURS 3 TRINN 07 TID
@AND VST80_K3_LUT_UTE
MOV(021) #7 VST80_K3_STATUS
; rung 3: VASK OK
LD P_On
AND K3_TR22_TID_S
MOV(021) #0 VST80_K3_STATUS

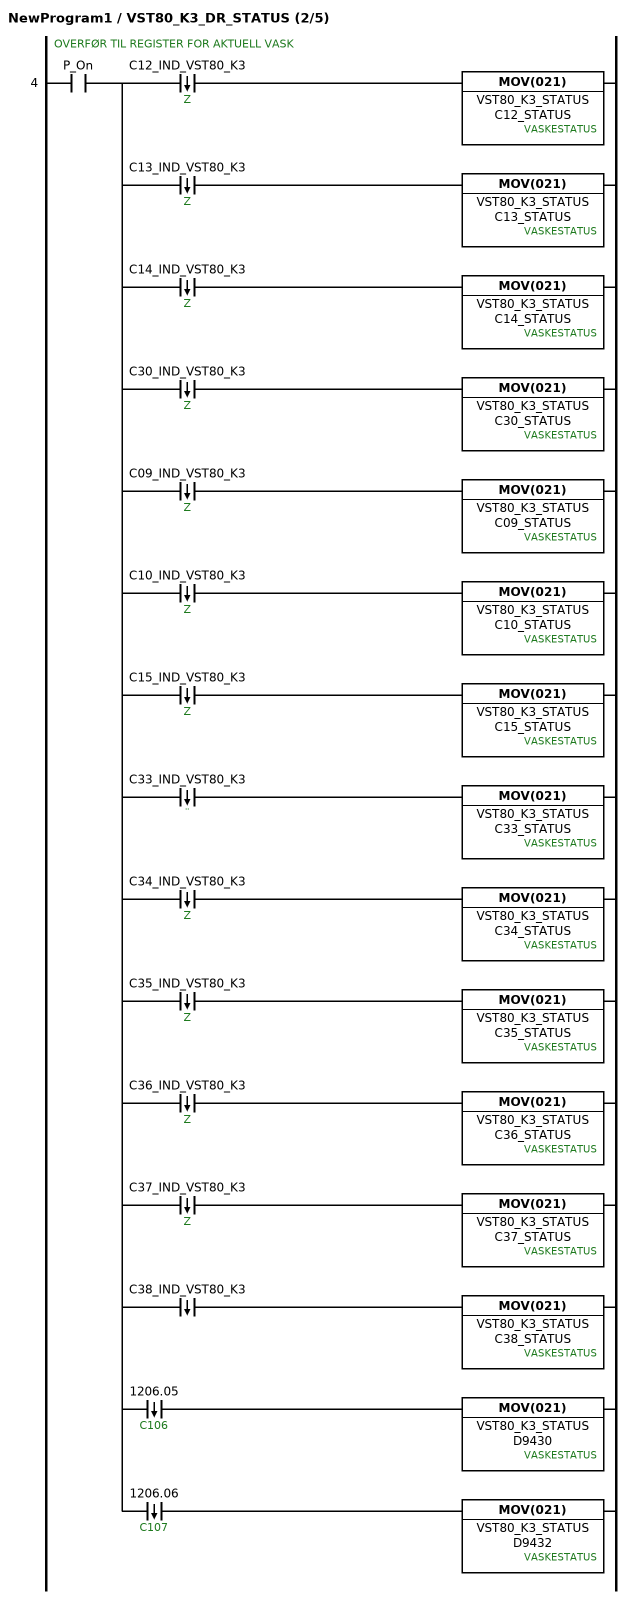
; rung 4: OVERFØR TIL REGISTER FOR AKTUELL VASK
LD P_On
OUT TR0
%AND C12_IND_VST80_K3  ; Z
MOV(021) VST80_K3_STATUS C12_STATUS  ; VASKESTATUS
LD TR0
%AND C13_IND_VST80_K3  ; Z
MOV(021) VST80_K3_STATUS C13_STATUS  ; VASKESTATUS
LD TR0
%AND C14_IND_VST80_K3  ; Z
MOV(021) VST80_K3_STATUS C14_STATUS  ; VASKESTATUS
LD TR0
%AND C30_IND_VST80_K3  ; Z
MOV(021) VST80_K3_STATUS C30_STATUS  ; VASKESTATUS
LD TR0
%AND C09_IND_VST80_K3  ; Z
MOV(021) VST80_K3_STATUS C09_STATUS  ; VASKESTATUS
LD TR0
%AND C10_IND_VST80_K3  ; Z
MOV(021) VST80_K3_STATUS C10_STATUS  ; VASKESTATUS
LD TR0
%AND C15_IND_VST80_K3  ; Z
MOV(021) VST80_K3_STATUS C15_STATUS  ; VASKESTATUS
LD TR0
%AND C33_IND_VST80_K3  ; ¨
MOV(021) VST80_K3_STATUS C33_STATUS  ; VASKESTATUS
LD TR0
%AND C34_IND_VST80_K3  ; Z
MOV(021) VST80_K3_STATUS C34_STATUS  ; VASKESTATUS
LD TR0
%AND C35_IND_VST80_K3  ; Z
MOV(021) VST80_K3_STATUS C35_STATUS  ; VASKESTATUS
LD TR0
%AND C36_IND_VST80_K3  ; Z
MOV(021) VST80_K3_STATUS C36_STATUS  ; VASKESTATUS
LD TR0
%AND C37_IND_VST80_K3  ; Z
MOV(021) VST80_K3_STATUS C37_STATUS  ; VASKESTATUS
LD TR0
%AND C38_IND_VST80_K3
MOV(021) VST80_K3_STATUS C38_STATUS  ; VASKESTATUS
LD TR0
%AND 1206.05  ; C106
MOV(021) VST80_K3_STATUS D9430  ; VASKESTATUS
LD TR0
%AND 1206.06  ; C107
MOV(021) VST80_K3_STATUS D9432  ; VASKESTATUS

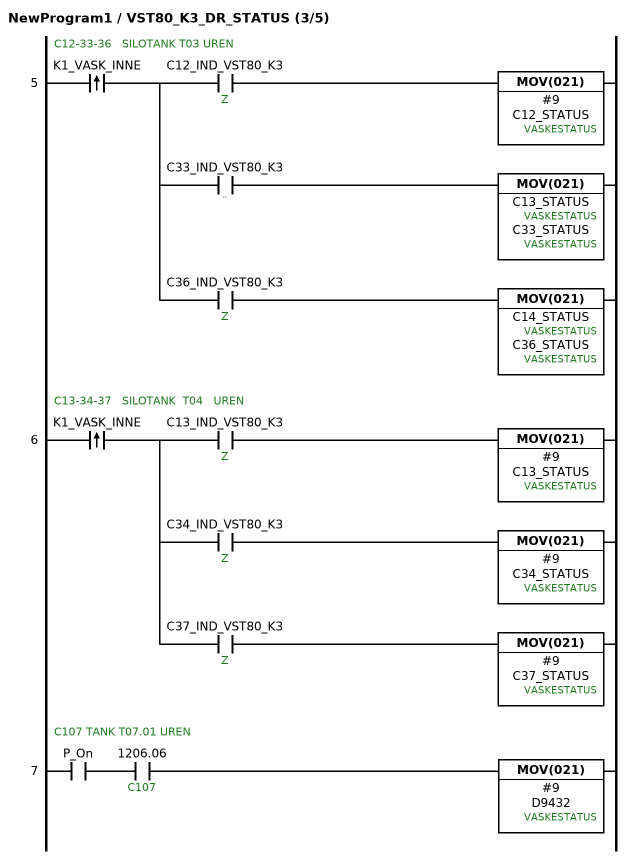
; rung 5: C12-33-36   SILOTANK T03 UREN
@LD K1_VASK_INNE
OUT TR0
AND C12_IND_VST80_K3  ; Z
MOV(021) #9 C12_STATUS  ; VASKESTATUS
LD TR0
AND C33_IND_VST80_K3  ; ¨
MOV(021) C13_STATUS C33_STATUS  ; VASKESTATUS
LD TR0
AND C36_IND_VST80_K3  ; Z
MOV(021) C14_STATUS C36_STATUS  ; VASKESTATUS
; rung 6: C13-34-37   SILOTANK  T04   UREN
@LD K1_VASK_INNE
OUT TR0
AND C13_IND_VST80_K3  ; Z
MOV(021) #9 C13_STATUS  ; VASKESTATUS
LD TR0
AND C34_IND_VST80_K3  ; Z
MOV(021) #9 C34_STATUS  ; VASKESTATUS
LD TR0
AND C37_IND_VST80_K3  ; Z
MOV(021) #9 C37_STATUS  ; VASKESTATUS
; rung 7: C107 TANK T07.01 UREN
LD P_On
AND 1206.06  ; C107
MOV(021) #9 D9432  ; VASKESTATUS

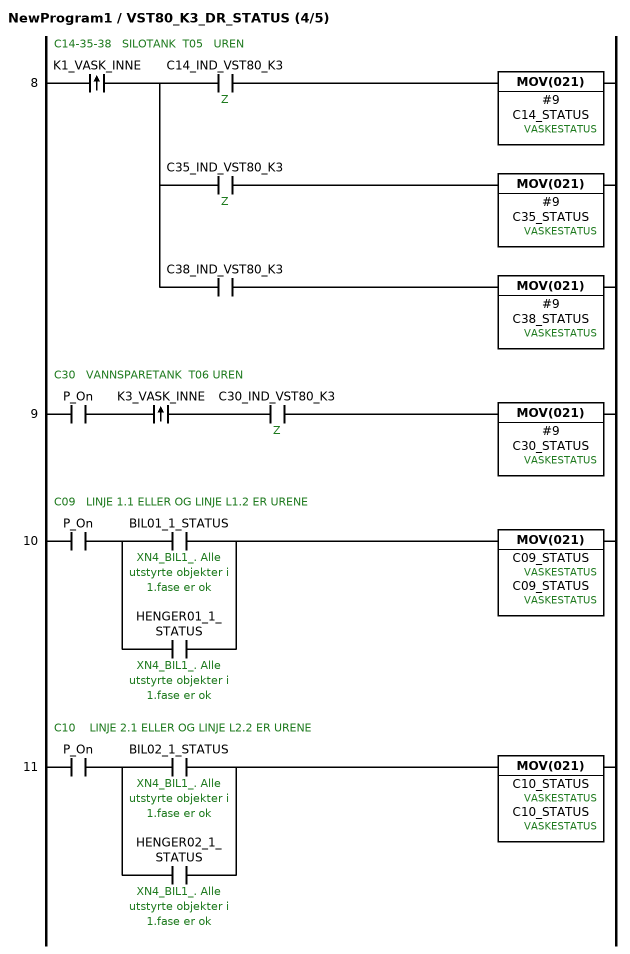
; rung 8: C14-35-38   SILOTANK  T05   UREN
@LD K1_VASK_INNE
OUT TR0
AND C14_IND_VST80_K3  ; Z
MOV(021) #9 C14_STATUS  ; VASKESTATUS
LD TR0
AND C35_IND_VST80_K3  ; Z
MOV(021) #9 C35_STATUS  ; VASKESTATUS
LD TR0
AND C38_IND_VST80_K3
MOV(021) #9 C38_STATUS  ; VASKESTATUS
; rung 9: C30   VANNSPARETANK  T06 UREN
LD P_On
@AND K3_VASK_INNE
AND C30_IND_VST80_K3  ; Z
MOV(021) #9 C30_STATUS  ; VASKESTATUS
; rung 10: C09   LINJE 1.1 ELLER OG LINJE L1.2 ER URENE
LD P_On
LD BIL01_1_STATUS  ; XN4_BIL1_. Alle utstyrte objekter i 1.fase er ok
OR HENGER01_1_STATUS  ; XN4_BIL1_. Alle utstyrte objekter i 1.fase er ok
ANDLD
MOV(021) C09_STATUS C09_STATUS  ; VASKESTATUS
; rung 11: C10    LINJE 2.1 ELLER OG LINJE L2.2 ER URENE
LD P_On
LD BIL02_1_STATUS  ; XN4_BIL1_. Alle utstyrte objekter i 1.fase er ok
OR HENGER02_1_STATUS  ; XN4_BIL1_. Alle utstyrte objekter i 1.fase er ok
ANDLD
MOV(021) C10_STATUS C10_STATUS  ; VASKESTATUS

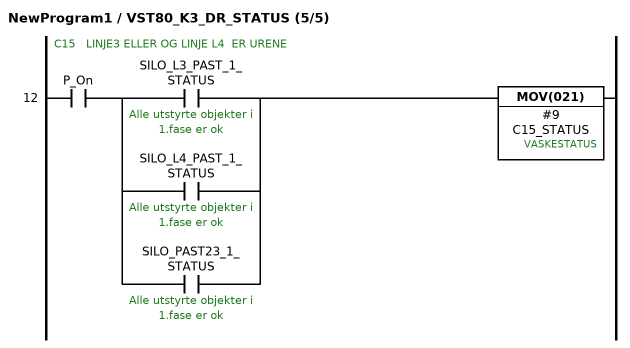
; rung 12: C15   LINJE3 ELLER OG LINJE L4  ER URENE
LD P_On
LD SILO_L3_PAST_1_STATUS  ; Alle utstyrte objekter i 1.fase er ok
OR SILO_L4_PAST_1_STATUS  ; Alle utstyrte objekter i 1.fase er ok
OR SILO_PAST23_1_STATUS  ; Alle utstyrte objekter i 1.fase er ok
ANDLD
MOV(021) #9 C15_STATUS  ; VASKESTATUS

### Section VST80_K3_FUNKSJON
; Dette programmet styrer kommandoene til vaskestasjonen.

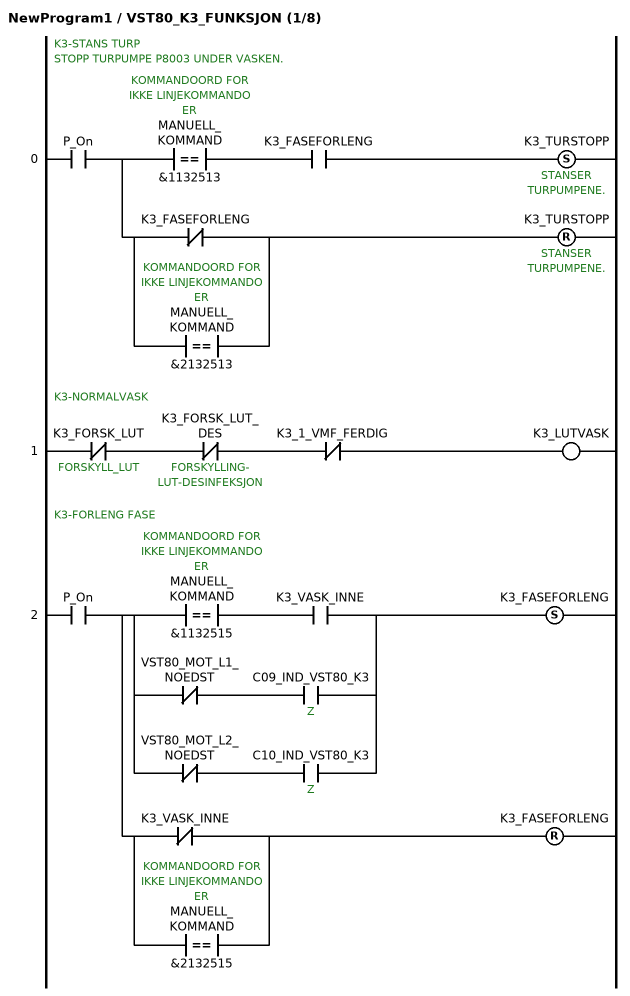
; rung 0: K3-STANS TURP / STOPP TURPUMPE P8003 UNDER VASKEN.
LD P_On
OUT TR0
AND=L(301) MANUELL_KOMMAND &1132513  ; KOMMANDOORD FOR IKKE LINJEKOMMANDOER
AND K3_FASEFORLENG
SET K3_TURSTOPP  ; STANSER TURPUMPENE.
LD TR0
LDNOT K3_FASEFORLENG
OR=L(301) MANUELL_KOMMAND &2132513  ; KOMMANDOORD FOR IKKE LINJEKOMMANDOER
ANDLD
RSET K3_TURSTOPP  ; STANSER TURPUMPENE.
; rung 1: K3-NORMALVASK
LDNOT K3_FORSK_LUT  ; FORSKYLL_LUT
ANDNOT K3_FORSK_LUT_DES  ; FORSKYLLING- LUT-DESINFEKSJON
ANDNOT K3_1_VMF_FERDIG
OUT K3_LUTVASK
; rung 2: K3-FORLENG FASE
LD P_On
OUT TR0
LD=L(301) MANUELL_KOMMAND &1132515  ; KOMMANDOORD FOR IKKE LINJEKOMMANDOER
AND K3_VASK_INNE
LDNOT VST80_MOT_L1_NOEDST
AND C09_IND_VST80_K3  ; Z
ORLD
LDNOT VST80_MOT_L2_NOEDST
AND C10_IND_VST80_K3  ; Z
ORLD
ANDLD
SET K3_FASEFORLENG
LD TR0
LDNOT K3_VASK_INNE
OR=L(301) MANUELL_KOMMAND &2132515  ; KOMMANDOORD FOR IKKE LINJEKOMMANDOER
ANDLD
RSET K3_FASEFORLENG

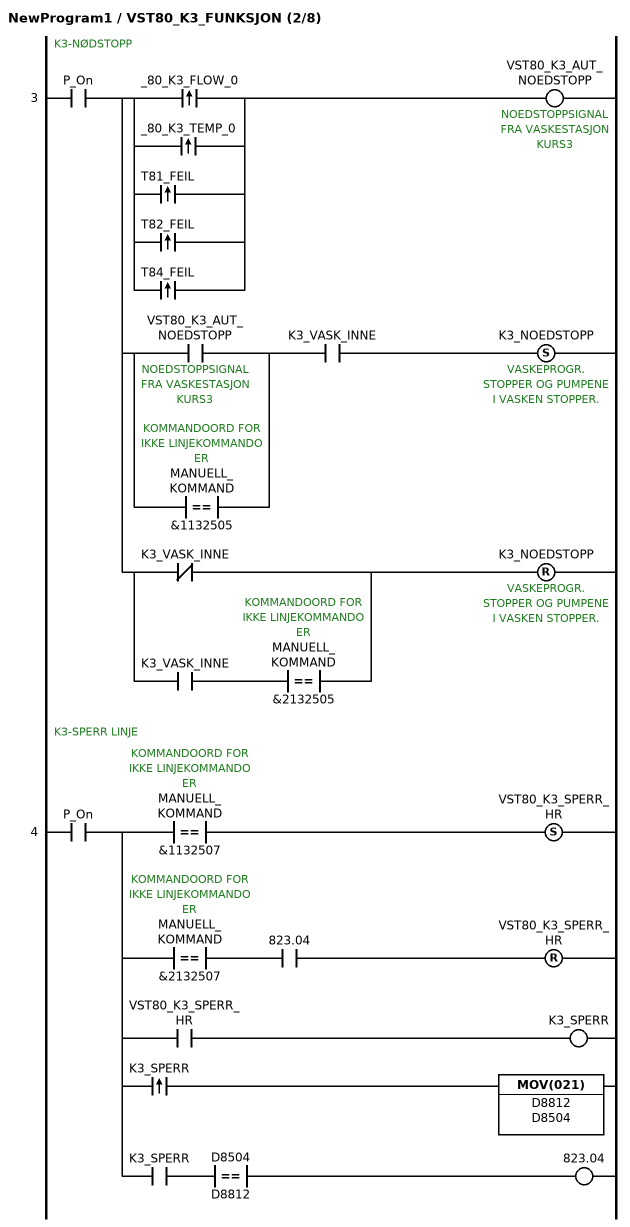
; rung 3: K3-NØDSTOPP
LD P_On
OUT TR0
@LD _80_K3_FLOW_0
@OR _80_K3_TEMP_0
@OR T81_FEIL
@OR T82_FEIL
@OR T84_FEIL
ANDLD
OUT VST80_K3_AUT_NOEDSTOPP  ; NOEDSTOPPSIGNAL FRA VASKESTASJON KURS3
LD TR0
LD VST80_K3_AUT_NOEDSTOPP  ; NOEDSTOPPSIGNAL FRA VASKESTASJON KURS3
OR=L(301) MANUELL_KOMMAND &1132505  ; KOMMANDOORD FOR IKKE LINJEKOMMANDOER
ANDLD
AND K3_VASK_INNE
SET K3_NOEDSTOPP  ; VASKEPROGR. STOPPER OG PUMPENE I VASKEN STOPPER.
LD TR0
LDNOT K3_VASK_INNE
LD K3_VASK_INNE
AND=L(301) MANUELL_KOMMAND &2132505  ; KOMMANDOORD FOR IKKE LINJEKOMMANDOER
ORLD
ANDLD
RSET K3_NOEDSTOPP  ; VASKEPROGR. STOPPER OG PUMPENE I VASKEN STOPPER.
; rung 4: K3-SPERR LINJE
LD P_On
OUT TR0
AND=L(301) MANUELL_KOMMAND &1132507  ; KOMMANDOORD FOR IKKE LINJEKOMMANDOER
SET VST80_K3_SPERR_HR
LD TR0
AND=L(301) MANUELL_KOMMAND &2132507  ; KOMMANDOORD FOR IKKE LINJEKOMMANDOER
AND 823.04
RSET VST80_K3_SPERR_HR
LD TR0
AND VST80_K3_SPERR_HR
OUT K3_SPERR
LD TR0
@AND K3_SPERR
MOV(021) D8812 D8504
LD TR0
AND K3_SPERR
AND=(300) D8504 D8812
OUT 823.04

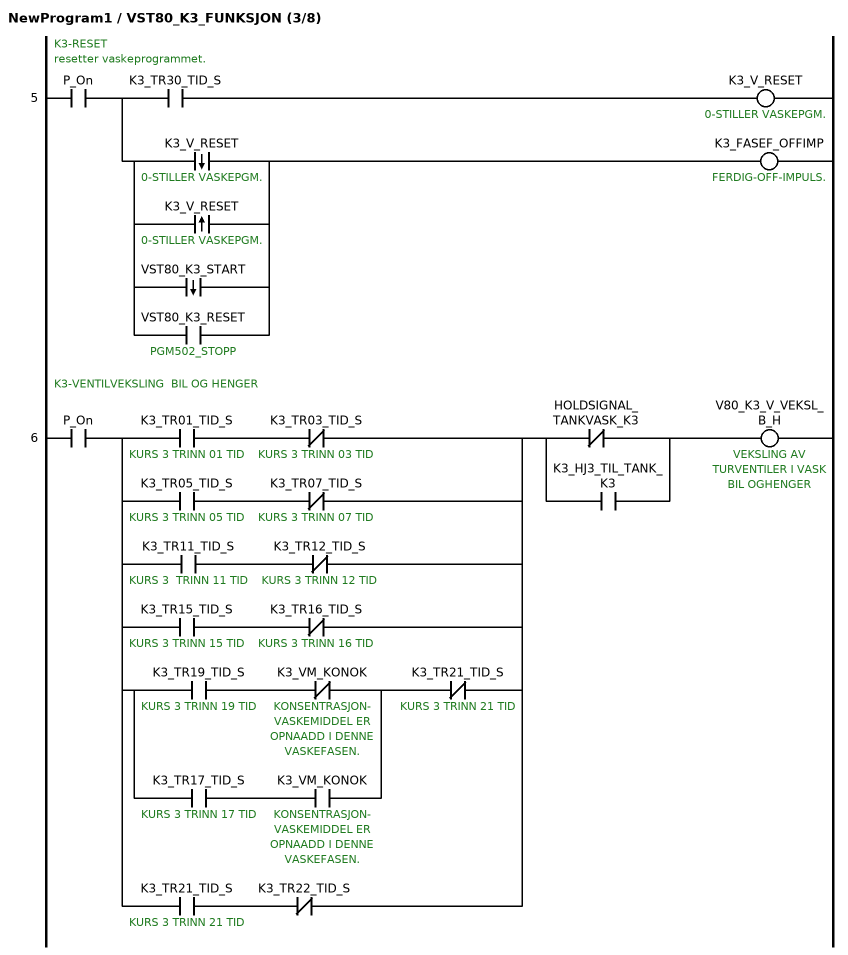
; rung 5: K3-RESET / resetter vaskeprogrammet.
LD P_On
OUT TR0
AND K3_TR30_TID_S
OUT K3_V_RESET  ; 0-STILLER VASKEPGM.
LD TR0
%LD K3_V_RESET  ; 0-STILLER VASKEPGM.
@OR K3_V_RESET  ; 0-STILLER VASKEPGM.
%OR VST80_K3_START
OR VST80_K3_RESET  ; PGM502_STOPP
ANDLD
OUT K3_FASEF_OFFIMP  ; FERDIG-OFF-IMPULS.
; rung 6: K3-VENTILVEKSLING  BIL OG HENGER
LD P_On
LD K3_TR01_TID_S  ; KURS 3 TRINN 01 TID
ANDNOT K3_TR03_TID_S  ; KURS 3 TRINN 03 TID
LD K3_TR05_TID_S  ; KURS 3 TRINN 05 TID
ANDNOT K3_TR07_TID_S  ; KURS 3 TRINN 07 TID
ORLD
LD K3_TR11_TID_S  ; KURS 3  TRINN 11 TID
ANDNOT K3_TR12_TID_S  ; KURS 3 TRINN 12 TID
ORLD
LD K3_TR15_TID_S  ; KURS 3 TRINN 15 TID
ANDNOT K3_TR16_TID_S  ; KURS 3 TRINN 16 TID
ORLD
LD K3_TR19_TID_S  ; KURS 3 TRINN 19 TID
ANDNOT K3_VM_KONOK  ; KONSENTRASJON-VASKEMIDDEL ER OPNAADD I DENNE VASKEFASEN.
LD K3_TR17_TID_S  ; KURS 3 TRINN 17 TID
AND K3_VM_KONOK  ; KONSENTRASJON-VASKEMIDDEL ER OPNAADD I DENNE VASKEFASEN.
ORLD
ANDNOT K3_TR21_TID_S  ; KURS 3 TRINN 21 TID
ORLD
LD K3_TR21_TID_S  ; KURS 3 TRINN 21 TID
ANDNOT K3_TR22_TID_S
ORLD
ANDLD
LDNOT HOLDSIGNAL_TANKVASK_K3
OR K3_HJ3_TIL_TANK_K3
ANDLD
OUT V80_K3_V_VEKSL_B_H  ; VEKSLING AV TURVENTILER I VASK BIL OGHENGER

